// TIA Portal V20 export
FUNCTION "FIT101_Liter" : Void   // FC26, FBD
{ S7_Optimized_Access := 'TRUE' }
// stored: SetENOAutomatically false
BEGIN

REGION Network 1: Channel input
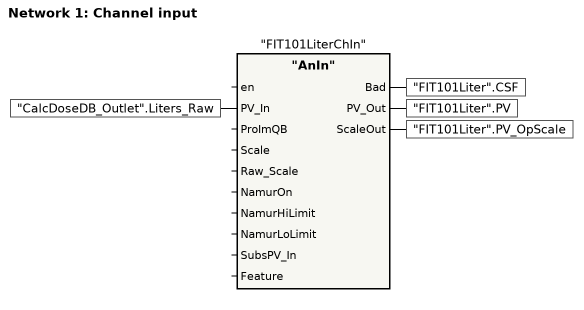
   "FIT101LiterChIn"(PV_In := "CalcDoseDB_Outlet".Liters_Raw,   // "AnIn"
                     Bad => "FIT101Liter".CSF,
                     PV_Out => "FIT101Liter".PV,
                     ScaleOut => "FIT101Liter".PV_OpScale);
END_REGION

REGION Network 2: MonAnL
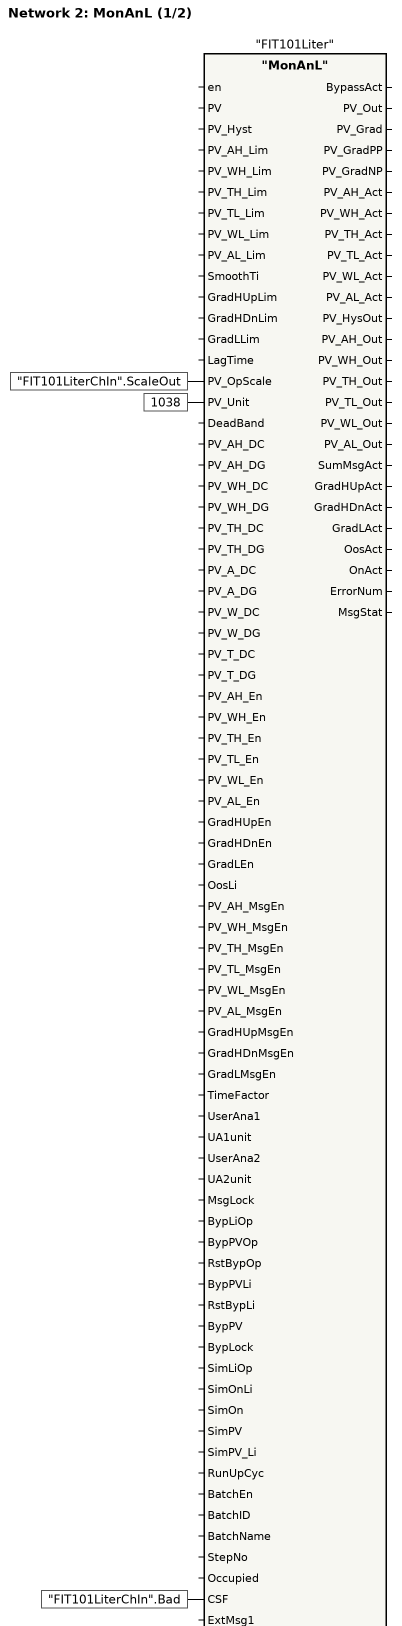
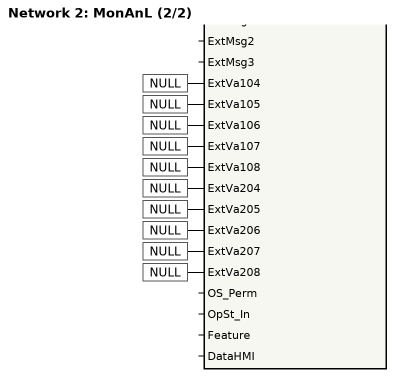
   "FIT101Liter"(PV_OpScale := "FIT101LiterChIn".ScaleOut,   // "MonAnL"
                 PV_Unit := 1038,
                 CSF := "FIT101LiterChIn".Bad,
                 ExtVa104 := NULL,
                 ExtVa105 := NULL,
                 ExtVa106 := NULL,
                 ExtVa107 := NULL,
                 ExtVa108 := NULL,
                 ExtVa204 := NULL,
                 ExtVa205 := NULL,
                 ExtVa206 := NULL,
                 ExtVa207 := NULL,
                 ExtVa208 := NULL);
END_REGION

REGION Network 3: MTP
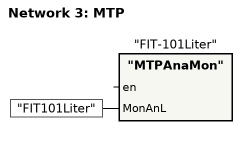
   "FIT-101Liter"(MonAnL := "FIT101Liter");   // "MTPAnaMon"
END_REGION
END_FUNCTION
